Omron Sysmac Studio project Arith (Sysmac Studio 1.65.0.64007, StandardProject)

# Controller new_Controller_0: NX1P2-1040DT1 version 1.69
Task PrimaryTask (priority 4, period or condition 2000): Program0

VAR_GLOBAL
    BIO_Input_Bit_00 : BOOL;  (* at BuiltInIO://cpu/#0/Input_Bit_00 *)
    BIO_Input_Bit_01 : BOOL;  (* at BuiltInIO://cpu/#0/Input_Bit_01 *)
    BIO_Input_Bit_02 : BOOL;  (* at BuiltInIO://cpu/#0/Input_Bit_02 *)
    BIO_Input_Bit_03 : BOOL;  (* at BuiltInIO://cpu/#0/Input_Bit_03 *)
    BIO_Output_Bit_00 : BOOL;  (* at BuiltInIO://cpu/#0/Output_Bit_00 *)
    IN_StartBut : BOOL;
    IN_StopBut : BOOL;
    IN_OptikSens : BOOL;
    IN_ResetBut : BOOL;
    OUT_Konveyor_Start : BOOL;
    IN_Konveyor_Start : BOOL;
END_VAR

PROGRAM Program0
VAR
    sayac : INT;
END_VAR
VAR_EXTERNAL
    BIO_Input_Bit_00 : BOOL;
    IN_StartBut : BOOL;
    BIO_Input_Bit_01 : BOOL;
    IN_StopBut : BOOL;
    BIO_Input_Bit_02 : BOOL;
    IN_OptikSens : BOOL;
    BIO_Input_Bit_03 : BOOL;
    IN_ResetBut : BOOL;
    OUT_Konveyor_Start : BOOL;
    BIO_Output_Bit_00 : BOOL;
    IN_Konveyor_Start : BOOL;
END_VAR
VAR
    _e1 : R_TRIG;
    _e2 : R_TRIG;
END_VAR

(* Section KoliSayma: ladder, written here as Structured Text *)

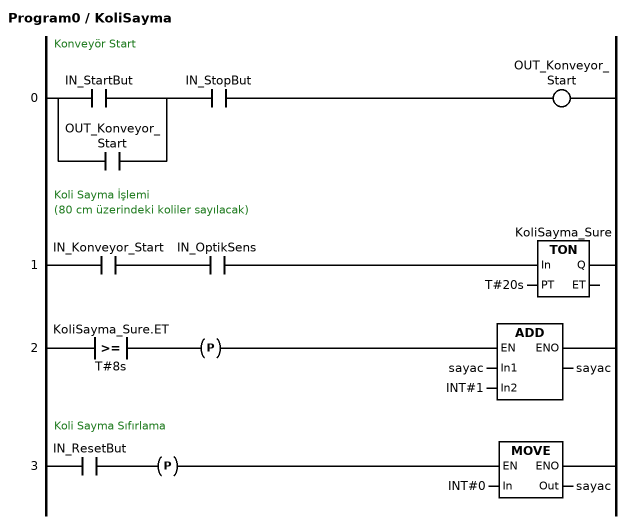
(* Rung 0: Konveyör Start *)
OUT_Konveyor_Start := (IN_StartBut OR OUT_Konveyor_Start) AND IN_StopBut;
(* Rung 1: Koli Sayma İşlemi / (80 cm üzerindeki koliler sayılacak) *)
KoliSayma_Sure(In := IN_Konveyor_Start AND IN_OptikSens, PT := T#20s);
(* Rung 2 *)
_e1(CLK := KoliSayma_Sure.ET >= T#8s);
IF _e1.Q THEN sayac := sayac + INT#1; END_IF;
(* Rung 3: Koli Sayma Sıfırlama *)
_e2(CLK := IN_ResetBut);
IF _e2.Q THEN sayac := INT#0; END_IF;

(* Section InOut: ladder, written here as Structured Text *)

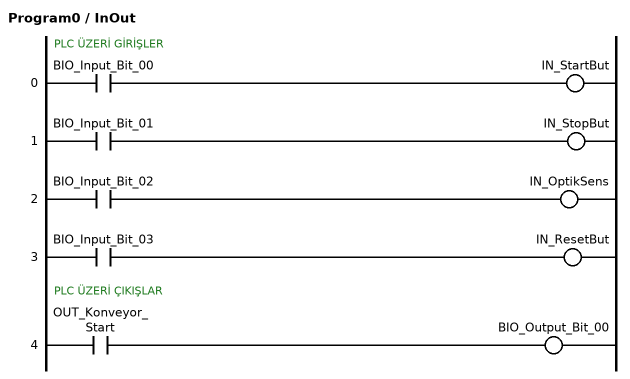
(* Rung 0: PLC ÜZERİ GİRİŞLER *)
IN_StartBut := BIO_Input_Bit_00;
(* Rung 1 *)
IN_StopBut := BIO_Input_Bit_01;
(* Rung 2 *)
IN_OptikSens := BIO_Input_Bit_02;
(* Rung 3 *)
IN_ResetBut := BIO_Input_Bit_03;
(* Rung 4: PLC ÜZERİ ÇIKIŞLAR *)
BIO_Output_Bit_00 := OUT_Konveyor_Start;
END_PROGRAM